(* Logix 5000 project; controller Ex_2_13 Emulate 5570 rev 33.11; software revision 33.00 *)
// Filling water into jerrycans

TASK MainTask (continuous, watchdog 500 ms) : MainProgram

MODULES
   Local : Emulate 5570 (ICP 4, rev 33.11)
END_MODULES

VAR_GLOBAL   (* controller tags *)
   B1 : BOOL;   // Sesnor B1
   B2 : BOOL;   // Sensor B2
   B5 : BOOL;   // Sensor B5
   M1 : BOOL;   // Conveyor Motor M1
   Q1 : BOOL;   // Eelctric Water Valve
END_VAR

PROGRAM MainProgram   (* main routine MainRoutine *)

ROUTINE MainRoutine   (* ladder *)
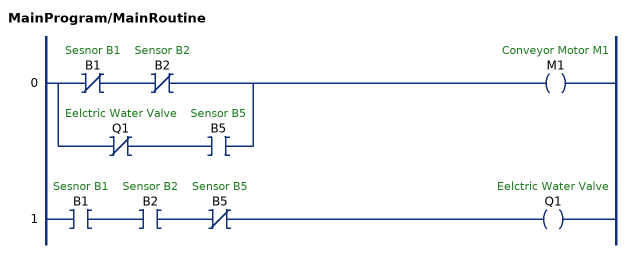
   0: [XIO(B1) XIO(B2) ,XIO(Q1) XIC(B5) ]OTE(M1);
   1: XIC(B1)XIC(B2)XIO(B5)OTE(Q1);
END_ROUTINE
END_PROGRAM
